// TIA Portal V19 export
TYPE "C501_STU_SME_TYPIC"
   STRUCT
      VGV_L { ExternalAccessible := 'False'; ExternalVisible := 'False'; ExternalWritable := 'False'} : USInt;   // Vrijgave detectie debiet te laag
   END_STRUCT;
END_TYPE
